FUNCTION_BLOCK ABSTRACT fb_MessageData IMPLEMENTS I_MessageData
VAR CONSTANT
{attribute 'hide'}
  STR_LEN       : UDINT := 524_288;
END_VAR
VAR
  _eCheck       : E_MESSAGE_CHECK;            // pointer check state

  _pFileRoot    : POINTER TO STRING(255);     // you decide (example in GVL_MSG.LOG_FILE)
  _pDirRoot     : POINTER TO STRING(255);     // see GVL_MSG.LOG_DIR

  _nMsgIndex    : REFERENCE TO UINT;          // Hypnos IS the only one in the village, if there are more you need more villages
  _nErrIndex    : REFERENCE TO UINT;          // Thanatos, Hypnos stern and more serious brother

  _dtLocalTime  : POINTER TO DT;
  _pMsgList     : POINTER TO ARRAY[1..GVL_MSG_XTS.MAX_MESSAGE] OF ST_Message; // attach your list here

	_rtrigReset   : Tc2_Standard.R_TRIG;
	_aWriteList   : ARRAY[1..GVL_MSG_XTS.MAX_MESSAGE] OF ST_Message;
	_sWriteData   : STRING(STR_LEN);
	_sNewLine     : STRING := '$N';
	_sTab         : STRING := '$T';
	_iCount, 
	_iStart, 
	_iEnd         : UINT;

	_fbCreateDir  : Tc2_System.FB_CreateDir;
	_sTmp         : STRING(256);
	_sFilename    : STRING(256);
	_sFolderDate  : STRING;
	_bFileCreated : BOOL;

	_fbFileOpen   : Tc2_System.FB_FileOpen;
	_fbFileWrite  : Tc2_System.FB_FileWrite;
	_fbFileClose  : Tc2_System.FB_FileClose;
END_VAR

METHOD Builder : BOOL // string concat for length > 255
VAR_INPUT
  pInString   : POINTER TO STRING;
  pOutString  : POINTER TO STRING(STR_LEN);
  Length      : UINT;
END_VAR
VAR
  Counter     : UDINT;
  pInWork     : POINTER TO BYTE;
  pOutWork    : POINTER TO BYTE;
END_VAR
pOutWork := pOutString;
pInWork := pInString;
Counter := 0;

(*check termination*)
WHILE (pOutWork^ <> 0) AND
      (Counter < STR_LEN+1)
DO
  Counter := Counter + 1;
  pOutWork := pOutWork + 1;
END_WHILE

(* append only if data fits into output *)
IF (Counter + Length < STR_LEN+1)
THEN

  (* append data *)
  FOR Counter := 1 TO Length
  DO
    pOutWork^ := pInWork^;
    pOutWork := pOutWork + 1;
    pInWork := pInWork + 1;
  END_FOR

  (* terminate *)
  pOutWork := pOutWork + 1;
  pOutWork^ := 0;
END_IF
END_METHOD

METHOD Check : BOOL
VAR_INPUT
END_VAR

IF NOT (_dtLocalTime <> 0)
THEN
  _eCheck       := E_MESSAGE_CHECK.POINTER_TIME_INVALID;
  RETURN;
END_IF

IF NOT (_pMsgList <> 0)
THEN
  _eCheck       := E_MESSAGE_CHECK.POINTER_LIST_INVALID;
  RETURN;
END_IF

IF NOT (_pFileRoot <> 0)
THEN
  _eCheck       := E_MESSAGE_CHECK.POINTER_ROOT_FILE_INVALID;
  RETURN;
END_IF

IF NOT (_pDirRoot <> 0)
THEN
  _eCheck       := E_MESSAGE_CHECK.POINTER_ROOT_DIR_INVALID;
  RETURN;
END_IF

IF NOT __ISVALIDREF(_nMsgIndex)
THEN
  _eCheck       := E_MESSAGE_CHECK.POINTER_MSG_IDX_INVALID;
  RETURN;
END_IF

IF NOT __ISVALIDREF(_nErrIndex)
THEN
  _eCheck       := E_MESSAGE_CHECK.POINTER_ERR_IDX_INVALID;
  RETURN;
END_IF


_eCheck         := E_MESSAGE_CHECK.CHECK_DONE;
Check           := TRUE;
END_METHOD

METHOD Device_to_String : string
VAR_INPUT
  eMsgDevice    : e_Device;
END_VAR
VAR
  sId                 : STRING := '_ID_';
  nId                 : UDINT;
END_VAR
IF (eMsgDevice < e_device.General)
THEN
  // below general case
  nId := TO_UDINT(eMsgDevice);
  //sId := concat(sId, TO_STRING(nId));

  //Device_to_String := concat(TO_STRING(eMsgDevice), sId);
  Device_to_String := TO_STRING(eMsgDevice);

ELSE
  IF (eMsgDevice >= e_Device.DataProduct)
  THEN
    nId := eMsgDevice MOD e_Device.DataProduct;
    sId := concat(sId, TO_STRING(nId));
 
    Device_to_String := concat(TO_STRING(e_Device.DataProduct), sId);

  ELSIF (eMsgDevice >= e_Device.Application)
  THEN
    nId := eMsgDevice MOD e_Device.Application;
    sId := concat(sId, TO_STRING(nId));
 
    Device_to_String := concat(TO_STRING(e_Device.Application), sId);

  ELSIF (eMsgDevice >= e_Device.TicketListCtrl)
  THEN
    nId := eMsgDevice MOD e_Device.TicketListCtrl;
    sId := concat(sId, TO_STRING(nId));
 
    Device_to_String := concat(TO_STRING(e_Device.TicketListCtrl), sId);

  ELSIF (eMsgDevice >= e_Device.ProcessListCtrl)
  THEN
    nId := eMsgDevice MOD e_Device.ProcessListCtrl;
    sId := concat(sId, TO_STRING(nId));
 
    Device_to_String := concat(TO_STRING(e_Device.ProcessListCtrl), sId);

  ELSIF (eMsgDevice >= e_Device.Process)
  THEN
    nId := eMsgDevice MOD e_Device.Process;
    sId := concat(sId, TO_STRING(nId));
 
    Device_to_String := concat(TO_STRING(e_Device.Process), sId);

  ELSIF (eMsgDevice >= e_Device.MetricsAxis)
  THEN
    nId := eMsgDevice MOD e_Device.MetricsAxis;
    sId := concat(sId, TO_STRING(nId));
 
    Device_to_String := concat(TO_STRING(e_device.MetricsAxis), sId);

  ELSIF (eMsgDevice >= e_Device.MetricsXts)
  THEN
    nId := eMsgDevice MOD e_Device.MetricsXts;
    sId := concat(sId, TO_STRING(nId));
 
    Device_to_String := concat(TO_STRING(e_device.MetricsXts), sId);

  ELSIF (eMsgDevice >= e_device.XfcAxis)
  THEN
    nId := eMsgDevice MOD e_device.XfcAxis;
    sId := concat(sId, TO_STRING(nId));
 
    Device_to_String := concat(TO_STRING(e_device.XfcAxis), sId);

  ELSIF (eMsgDevice >= e_device.Axis)
  THEN
    nId := eMsgDevice MOD e_device.Axis;
    sId := concat(sId, TO_STRING(nId));
 
    Device_to_String := concat(TO_STRING(e_device.Axis), sId);

  ELSIF (eMsgDevice >= e_device.NciChannelCtrl)
  THEN
    nId := eMsgDevice MOD e_device.NciChannelCtrl;
    sId := concat(sId, TO_STRING(nId));
 
    Device_to_String := concat(TO_STRING(e_device.NciChannelCtrl), sId);

  ELSIF (eMsgDevice >= e_device.NciChannel)
  THEN
    nId := eMsgDevice MOD e_device.NciChannel;
    sId := concat(sId, TO_STRING(nId));
 
    Device_to_String := concat(TO_STRING(e_device.NciChannel), sId);

  ELSIF (eMsgDevice >= e_Device.Camming)
  THEN
    nId := eMsgDevice MOD e_Device.Camming;
    sId := concat(sId, TO_STRING(nId));
 
    Device_to_String := concat(TO_STRING(e_device.Camming), sId);

  ELSIF (eMsgDevice >= e_Device.XtsStation)
  THEN
    nId := eMsgDevice MOD e_Device.XtsStation;
    sId := concat(sId, TO_STRING(nId));
 
    Device_to_String := concat(TO_STRING(e_device.XtsStation), sId);

  ELSIF (eMsgDevice >= e_Device.XfcTouchProbe)
  THEN
    nId := eMsgDevice MOD e_Device.XfcTouchProbe;
    sId := concat(sId, TO_STRING(nId));
 
    Device_to_String := concat(TO_STRING(e_device.XfcTouchProbe), sId);

  ELSIF (eMsgDevice >= e_Device.XfcTriggerBox)
  THEN
    nId := eMsgDevice MOD e_Device.XfcTriggerBox;
    sId := concat(sId, TO_STRING(nId));
 
    Device_to_String := concat(TO_STRING(e_device.XfcTriggerBox), sId);

  ELSIF (eMsgDevice >= e_Device.XtsTransportUnit)
  THEN
    nId := eMsgDevice MOD e_Device.XtsTransportUnit;
    sId := concat(sId, TO_STRING(nId));
 
    Device_to_String := concat(TO_STRING(e_device.XtsTransportUnit), sId);

  ELSIF (eMsgDevice >= e_Device.MoverCtrl)
  THEN
    nId := eMsgDevice MOD e_Device.MoverCtrl;
    sId := concat(sId, TO_STRING(nId));
 
    Device_to_String := concat(TO_STRING(e_device.MoverCtrl), sId);

  ELSIF (eMsgDevice >= e_Device.Mover)
  THEN
    nId := eMsgDevice MOD e_Device.Mover;
    sId := concat(sId, TO_STRING(nId));
 
    Device_to_String := concat(TO_STRING(e_device.Mover), sId);

  ELSIF (eMsgDevice >= e_Device.XpuCtrl)
  THEN
    nId := eMsgDevice MOD e_Device.XpuCtrl;
    sId := concat(sId, TO_STRING(nId));
 
    Device_to_String := concat(TO_STRING(e_device.XpuCtrl), sId);

  ELSIF (eMsgDevice >= e_Device.Xpu)
  THEN
    nId := eMsgDevice MOD e_Device.Xpu;
    sId := concat(sId, TO_STRING(nId));
 
    Device_to_String := concat(TO_STRING(e_device.Xpu), sId);

  ELSIF (eMsgDevice >= e_Device.CaGroup)
  THEN
    nId := eMsgDevice MOD e_Device.CaGroup;
    sId := concat(sId, TO_STRING(nId));
 
    Device_to_String := concat(TO_STRING(e_device.CaGroup), sId);

  ELSIF (eMsgDevice >= e_Device.General)
  THEN
    nId := eMsgDevice MOD e_Device.General;
    //sId := concat(sId, TO_STRING(nId));
 
    Device_to_String := TO_STRING(e_device.General);

  ELSE
    Device_to_String := TO_STRING(eMsgDevice);
  END_IF
END_IF
END_METHOD

PROPERTY DirRoot : POINTER to string(255)
SET
_pDirRoot := DirRoot;
END_SET
END_PROPERTY

PROPERTY ErrorIndex : reference to uint
SET
_nErrIndex  REF= ErrorIndex;
END_SET
END_PROPERTY

PROPERTY FileRoot : pointer to string(255)
SET
_pFileRoot := FileRoot;
END_SET
END_PROPERTY

METHOD FolderDate : STRING
VAR_INPUT
	LocalTime   : POINTER TO DT;
END_VAR
VAR
	sTmp        : STRING;
END_VAR
IF NOT (LocalTime <> 0)
THEN
	FolderDate := 'NULL';
	RETURN;
END_IF

sTmp := DT_TO_STRING(LocalTime^);

// cut off #dt literal
sTmp := right(sTmp, len(sTmp)-3);

sTmp := replace(sTmp, '_', 1, 5);
sTmp := replace(sTmp, '_', 1, 8);

sTmp := left(sTmp,10);	// year_month_day

FolderDate := sTmp;
END_METHOD

PROPERTY LocalTime : pointer to DT
SET
_dtLocalTime := LocalTime;
END_SET
END_PROPERTY

PROPERTY MessageIndex : reference to uint
SET
_nMsgIndex   REF= MessageIndex;
END_SET
END_PROPERTY

PROPERTY MsgList : pointer to ARRAY[1..GVL_MSG_XTS.MAX_MESSAGE] OF st_message
SET
_pMsgList := MsgList;
END_SET
END_PROPERTY

METHOD StringLen : UINT // 	string length for len > 255
VAR_INPUT
  pInString		: POINTER TO STRING(STR_LEN);
END_VAR
VAR
	Counter			: UINT;
	pInWork			: POINTER TO BYTE;
END_VAR
pInWork := pInString;
Counter := 0;

WHILE (pInWork^ <> 0) AND
			(Counter < STR_LEN)
DO
	Counter := Counter + 1;
	pInWork := pInWork + 1;
END_WHILE

StringLen := Counter;
END_METHOD

METHOD WriteData  : e_progress
VAR_INPUT
  bExecute        : BOOL;
END_VAR
VAR_INST
  _eState         : e_progress;
  _bError         : BOOL;
  _nErrorId       : UDINT;
END_VAR
IF NOT bExecute
THEN
  _eState                     := E_PROGRESS.PROGRESS_INIT;
END_IF

CASE _eState 
OF

	E_PROGRESS.PROGRESS_INIT:
    _fbFileOpen(
        sPathName             := _sFilename, 
        nMode                 := FOPEN_MODEAPPEND OR FOPEN_MODEPLUS, 
        ePath                 := PATH_GENERIC, 
        bExecute              := FALSE, 
        tTimeout              := T#5S);

    _fbFileWrite(
        hFile                 := _fbFileOpen.hFile, 
        pWriteBuff            := ADR(_sWriteData), 
        cbWriteLen            := StringLen(ADR(_sWriteData)),
        bExecute              := FALSE, 
        tTimeout              := T#5S);

    _fbFileClose(
        hFile                 := _fbFileOpen.hFile, 
        bExecute              := FALSE, 
        tTimeout              := T#5S);


		IF bExecute
		THEN
      _nErrorId               := 0;
      _eState                 := E_PROGRESS.PROGRESS_BUSY;
		END_IF

	E_PROGRESS.PROGRESS_BUSY:
		_fbFileOpen(bExecute      := TRUE);

    IF _fbFileOpen.bError
    THEN
      _nErrorId               := _fbFileOpen.nErrId;
      _eState                 := E_PROGRESS.PROGRESS_ERROR;

		ELSIF _fbFileOpen.bBusy
		THEN
      _eState                 := E_PROGRESS.PROGRESS_PREPARE;
		END_IF

	E_PROGRESS.PROGRESS_PREPARE:
		_fbFileOpen(bExecute      := TRUE);
		IF NOT _fbFileOpen.bBusy
		THEN
		  _fbFileOpen(bExecute    := FALSE);
      _eState                 := E_PROGRESS.PROGRESS_STARTUP;
		END_IF

	E_PROGRESS.PROGRESS_STARTUP:
    _fbFileWrite(
        hFile                 := _fbFileOpen.hFile, 
        pWriteBuff            := ADR(_sWriteData), 
        cbWriteLen            := StringLen(ADR(_sWriteData)),
        bExecute              := TRUE, 
        tTimeout              := T#5S);

    IF _fbFileWrite.bError
    THEN
      _nErrorId               := _fbFileWrite.nErrId;
      _eState                 := E_PROGRESS.PROGRESS_ERROR;

		ELSIF _fbFileWrite.bBusy
		THEN
      _eState                 := E_PROGRESS.PROGRESS_CHECK;
		END_IF

	E_PROGRESS.PROGRESS_CHECK:
	  _fbFileWrite(bExecute     := TRUE);
		IF NOT _fbFileWrite.bBusy
		THEN
			_fbFileWrite(bExecute   := FALSE);
      _eState                 := E_PROGRESS.PROGRESS_OCCUPIED;
		END_IF

	E_PROGRESS.PROGRESS_OCCUPIED:
    _fbFileClose(
        hFile                 := _fbFileOpen.hFile, 
        bExecute              := TRUE, 
        tTimeout              := T#5S);

    IF _fbFileClose.bError
    THEN
      _nErrorId               := _fbFileClose.nErrId;
      _eState                 := E_PROGRESS.PROGRESS_ERROR;

		ELSIF _fbFileClose.bBusy
		THEN
      _eState                 := E_PROGRESS.PROGRESS_WORKING;
		END_IF

	E_PROGRESS.PROGRESS_WORKING:
    _fbFileClose(bExecute     := TRUE);
		IF NOT _fbFileClose.bBusy
		THEN
			_fbFileClose(bExecute   := FALSE);
      _eState                 := E_PROGRESS.PROGRESS_DONE;
		END_IF

END_CASE
CASE _eState
OF
  E_PROGRESS.PROGRESS_ERROR:
		_fbFileOpen (bExecute     := FALSE);
    _fbFileWrite(bExecute     := FALSE);
    _fbFileClose(bExecute     := FALSE);


END_CASE




WriteData                     := _eState;
END_METHOD

END_FUNCTION_BLOCK

(* stored: Version 1.1.0.1, ProductVersion 3.1.4026.18
   POU fb_MessageData: Id {cb8ad496-c9e3-4fb2-8dc7-4dc91b6a6f2d}, SpecialFunc None
   Folder methods: Id {287a4d29-6639-428c-aea8-52d8fb01790b}
   Folder properties: Id {a6c51d25-007d-41d8-ba61-13bf11666244}
   Method Builder: Id {04be8aaa-8316-4947-8184-69b641441e20}
   Method Check: Id {83de2011-150a-4d2a-94c5-1279228c4cba}
   Method Device_to_String: Id {f3e17cf0-bd04-48d4-acb3-86468a20329c}
   Property DirRoot: Id {7397fe37-0041-46ca-803c-f0222d19c8d7}
   Set Set: Id {92122c83-fc4a-4bda-97fd-a71f040ce274}
   Property ErrorIndex: Id {86b66e73-e80f-4556-8b0a-816c3404df55}
   Set Set: Id {5482dafd-b40d-4343-bb04-37805b132305}
   Property FileRoot: Id {d6de2757-e0df-464b-a162-cacc1b6bdb3d}
   Set Set: Id {7108b8fb-fc96-4838-8c31-c443544aad4a}
   Method FolderDate: Id {6be63320-fddb-4b4f-9db1-f5ca5528018c}
   Property LocalTime: Id {f651bcfe-d05f-47e1-b13f-4c3505347a64}
   Set Set: Id {7aff097a-64e1-4c25-823e-4e2f78f82768}
   Property MessageIndex: Id {2143a87e-4123-4fe9-9031-41726503bc50}
   Set Set: Id {9d407f6d-9268-4338-91af-524c55669750}
   Property MsgList: Id {78574afd-c9cb-4679-ae25-dbd5f9a9ae54}
   Set Set: Id {7d88d082-559f-4a6b-b0ff-94440fb4fde0}
   Method StringLen: Id {643ca8f7-a9e4-4425-bb86-0f8509d202ae}
   Method WriteData: Id {ec9b73b1-ecb3-44d9-883b-ae97dbd42464} *)
